// TIA Portal V17 export
// export: Created 2025-03-05T08:03:24.3570839Z, ExportSetting WithDefaults, DisplayName Totally Integrated Automation Portal, DisplayVersion V17 Update 8, DisplayName TIA Portal Openness, DisplayVersion V17 Update 8, DisplayName TIA Portal Version Control Interface, DisplayVersion V17, DisplayName SINAMICS Startdrive Advanced, DisplayVersion V17 SP2, DisplayName SINAMICS Startdrive G110M, G120, G120C, G120D, G120P, G115D, DisplayVersion V17 SP2, DisplayName SINAMICS Startdrive G130, G150, S120, S150, SINAMICS MV, S210, DisplayVersion V17 SP2, DisplayName STEP 7 Professional, DisplayVersion V17 Update 8, DisplayName SINUMERIK ONE STEP 7 Toolbox, DisplayVersion V17 Update 12, DisplayName SINUMERIK 840D sl STEP 7 Toolbox, DisplayVersion V17 Update 12, DisplayName STEP 7 Safety, DisplayVersion V17 Update 6, DisplayName WinCC Advanced, DisplayVersion V17 Update 8
DATA_BLOCK "DB22150_WP321_WEIGHT_CELLS"   // DB22150
VERSION : 0.1
// stored: AutoNumber false, DBAccessibleFromOPCUA true, DBAccessibleFromWebserver true, InstanceOfName FB22107_WP321_MUL_CALL, InstanceOfType FB
"FB22107_WP321_MUL_CALL"
   // VAR_INPUT
   //    SynchronizeAllDataFromSiwarexToDataBlockOnStartUp : Bool;
   // END_VAR
   // VAR_OUTPUT
   //    ArrayStartValue : Int;
   //    ArrayMaxValue : Int;
   // END_VAR
   // VAR
   //    WP321DR { S7_SetPoint := 'True'} : Array[0..7] of "WP321DR";
   //    FBStartUpTemp { S7_SetPoint := 'True'} : Array[0..7] of Bool;
   // END_VAR
BEGIN
END_DATA_BLOCK
